FUNCTION_BLOCK cfb_week_classifier
  (* Standard: 61499-2 *)
  (* Version 0.1, 2018-00-27, palme, DESKTOP-TGOEKBD *)
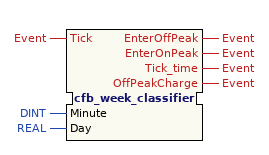
  EVENT_INPUT
    Tick;
  END_EVENT
  EVENT_OUTPUT
    EnterOffPeak;
    EnterOnPeak;
    Tick_time;
    OffPeakCharge;
  END_EVENT
  VAR_INPUT
    Minute : DINT;
    Day : REAL;
  END_VAR
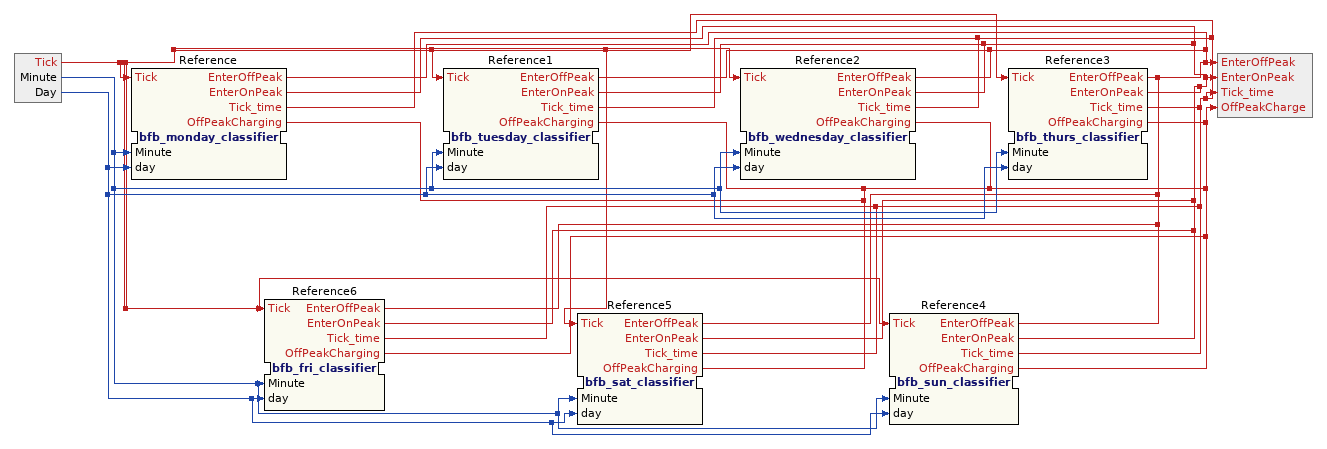
  FBS
    Reference : bfb_monday_classifier;
    Reference1 : bfb_tuesday_classifier;
    Reference2 : bfb_wednesday_classifier;
    Reference3 : bfb_thurs_classifier;
    Reference4 : bfb_sun_classifier;
    Reference5 : bfb_sat_classifier;
    Reference6 : bfb_fri_classifier;
  END_FBS
  EVENT_CONNECTIONS
    Tick TO Reference.Tick;
    Tick TO Reference1.Tick;
    Tick TO Reference2.Tick;
    Tick TO Reference3.Tick;
    Tick TO Reference6.Tick;
    Tick TO Reference5.Tick;
    Tick TO Reference4.Tick;
    Reference.EnterOffPeak TO EnterOffPeak;
    Reference1.EnterOffPeak TO EnterOffPeak;
    Reference2.EnterOffPeak TO EnterOffPeak;
    Reference3.EnterOffPeak TO EnterOffPeak;
    Reference6.EnterOffPeak TO EnterOffPeak;
    Reference5.EnterOffPeak TO EnterOffPeak;
    Reference4.EnterOffPeak TO EnterOffPeak;
    Reference.EnterOnPeak TO EnterOnPeak;
    Reference1.EnterOnPeak TO EnterOnPeak;
    Reference2.EnterOnPeak TO EnterOnPeak;
    Reference3.EnterOnPeak TO EnterOnPeak;
    Reference6.EnterOnPeak TO EnterOnPeak;
    Reference5.EnterOnPeak TO EnterOnPeak;
    Reference4.EnterOnPeak TO EnterOnPeak;
    Reference.Tick_time TO Tick_time;
    Reference1.Tick_time TO Tick_time;
    Reference2.Tick_time TO Tick_time;
    Reference3.Tick_time TO Tick_time;
    Reference6.Tick_time TO Tick_time;
    Reference5.Tick_time TO Tick_time;
    Reference4.Tick_time TO Tick_time;
    Reference.OffPeakCharging TO OffPeakCharge;
    Reference1.OffPeakCharging TO OffPeakCharge;
    Reference2.OffPeakCharging TO OffPeakCharge;
    Reference3.OffPeakCharging TO OffPeakCharge;
    Reference6.OffPeakCharging TO OffPeakCharge;
    Reference5.OffPeakCharging TO OffPeakCharge;
    Reference4.OffPeakCharging TO OffPeakCharge;
  END_CONNECTIONS
  DATA_CONNECTIONS
    Minute TO Reference4.Minute;
    Minute TO Reference5.Minute;
    Minute TO Reference6.Minute;
    Minute TO Reference.Minute;
    Minute TO Reference1.Minute;
    Minute TO Reference2.Minute;
    Minute TO Reference3.Minute;
    Day TO Reference4.day;
    Day TO Reference5.day;
    Day TO Reference6.day;
    Day TO Reference.day;
    Day TO Reference1.day;
    Day TO Reference2.day;
    Day TO Reference3.day;
  END_CONNECTIONS
END_FUNCTION_BLOCK
